{attribute 'qualified_only'}
{attribute 'strict'}
{attribute 'to_string'}
TYPE ePowerModes :
(
	DroopZeroStart 		:= 0,
	Droop				:= 1,
	Isochronous			:= 2
);
END_TYPE

(* stored: Version 1.1.0.1, ProductVersion 3.1.4026.18
   DUT ePowerModes: Id {cb37e4c4-f853-488e-8be0-e9eff17b66eb} *)
